Fanuc KAREL source: ko00081.KL

-- PROVISIONAL review KL for V1013-1; original PC SHA256 6ef2c4e9c6be315951f3650e716b090bddceb41698b3774d304d70da0ec2bde7
-- Incomplete behavior may be omitted. Consult companion uncertainty JSON. Do not deploy.
PROGRAM KO00081
%NOLOCKGROUP
BEGIN
  -- UNRESOLVED_PC offsets 5-12; opcodes 9D,23
  -- UNRESOLVED_PC offsets 17-66; opcodes 27,27,49,7E,AD,22,1C,22,31,7E,4A
  -- UNRESOLVED_PC offsets 71-75; opcodes 7F
END KO00081
